// TIA Portal V17 export
// export: Created 2022-03-12T16:05:29.9950523Z, ExportSetting WithDefaults, DisplayName Totally Integrated Automation Portal, DisplayVersion V17, DisplayName TIA Portal Openness, DisplayVersion V17, DisplayName TIA Portal Version Control Interface, DisplayVersion V17, DisplayName STEP 7 Professional, DisplayVersion V17, DisplayName STEP 7 Safety, DisplayVersion V17, DisplayName WinCC Advanced / Unified PC, DisplayVersion V17
DATA_BLOCK "RecipeCfg"   // DB1605
TITLE = CPG_RecipeCfg
{ S7_Optimized_Access := 'TRUE' }
AUTHOR : tech.team.motioncontrol@siemens.com
FAMILY : CPG
VERSION : 1.1
// Support: tech.team.motioncontrol@siemens.com
// stored: AutoNumber true, DBAccessibleFromOPCUA true, DBAccessibleFromWebserver true, IsOnlyStoredInLoadMemory false, IsRetainMemResEnabled false, IsWriteProtectedInAS false, MemoryReserve 0
   VAR
      setpoints_REAL { S7_SetPoint := 'True'} : Array[0.."CPG_NO_OF_SETPOINT_REAL_UPPER_LIM"] of "CPG_typeRecipeSetpoint_REAL";   // Array of setpoints of REAL
      setpoints_DINT { S7_SetPoint := 'True'} : Array[0.."CPG_NO_OF_SETPOINT_DINT_UPPER_LIM"] of "CPG_typeRecipeSetpoint_DINT";   // Array of setpoints of DINT
      setpoints_BOOL { S7_SetPoint := 'True'} : Array[0.."CPG_NO_OF_SETPOINT_BOOL_UPPER_LIM"] of "CPG_typeRecipeSetpoint_BOOL";   // Array of setpoints of BOOL
      setpoints_STRING { S7_SetPoint := 'True'} : Array[0.."CPG_NO_OF_SETPOINT_STRING_UPPER_LIM"] of "CPG_typeRecipeSetpoint_STRING";   // Array of setpoints of STRING
      recipeControl { S7_SetPoint := 'True'} : "CPG_typeRecipeControl";   // FB_Recipe_Control communicates to the setpoints via this tag
      recipeNames : Array[0.."CPG_NO_OF_RECIPE_UPPER_LIM"] of String[60];   // Array holding the names of all recipes
      recipeCumTimes : Array[0.."CPG_NO_OF_RECIPE_UPPER_LIM"] of Time;   // Array holding the cumulative time all recipes have been active
      recipeLastSaveTimes : Array[0.."CPG_NO_OF_RECIPE_UPPER_LIM"] of DTL;   // Array holding the last time each recipe was saved
   END_VAR
BEGIN
   setpoints_REAL[0].SetpointName[0] := 'LH 1 Length';
   setpoints_DINT[0].SetpointName[0] := 'DINT SP 0';
   setpoints_BOOL[0].SetpointName[0] := 'BOOL SP 0';
   setpoints_BOOL[0].SetpointName[1] := '';
   setpoints_BOOL[0].Text_True[0] := 'TRUE';
   setpoints_BOOL[0].Text_True[1] := '';
   setpoints_BOOL[0].Text_False[0] := 'FALSE';
   setpoints_STRING[0].RecipeValues[0] := 'a';
   setpoints_STRING[0].RecipeValues[1] := 'b';
   setpoints_STRING[0].RecipeValues[2] := 'c';
   setpoints_STRING[0].RecipeValues[3] := 'd';
   setpoints_STRING[0].RecipeValues[4] := 'e';
   setpoints_STRING[0].RecipeValues[5] := 'f';
   setpoints_STRING[0].RecipeValues[6] := 'g';
   setpoints_STRING[0].SetpointName[0] := 'STRING SP 0';
   recipeControl.CurrentRecipeID := 0;
   recipeControl.CurrentRecipeName := 'Recipe 0';
   recipeControl.RecipeID_A := 1;
   recipeControl.RecipeID_B := 2;
   recipeControl.RecipeID_C := 3;
   recipeNames[0] := 'Recipe 0';
   recipeNames[1] := 'Recipe 1';
   recipeNames[2] := 'Recipe 2';
   recipeNames[3] := 'Recipe 3';
   recipeNames[4] := 'Recipe 4';
   recipeNames[5] := 'Recipe 5';
   recipeNames[6] := 'Recipe 6';
   recipeNames[7] := 'Recipe 7';
   recipeNames[8] := 'Recipe 8';
   recipeNames[9] := 'Recipe 9';
   recipeNames[10] := 'Recipe 10';
   recipeNames[11] := 'Recipe 11';
   recipeNames[12] := 'Recipe 12';
   recipeNames[13] := 'Recipe 13';
   recipeNames[14] := 'Recipe 14';
   recipeNames[15] := 'Recipe 15';
   recipeNames[16] := 'Recipe 16';
   recipeNames[17] := 'Recipe 17';
   recipeNames[18] := 'Recipe 18';
   recipeNames[19] := 'Recipe 19';
   recipeNames[20] := 'Recipe 20';
   recipeLastSaveTimes[0..20] := DTL#2019-1-1-00:00:00;
END_DATA_BLOCK
